(* PLC project Unnamed, Unknown Unnamed 1 *)
(* stored: creationDateTime 2026-04-21T22:15:54, modificationDateTime 2026-04-21T22:15:54 *)

PROGRAM main
  VAR
    input AT %QW0 : INT;
    output AT %QW1 : INT;
  END_VAR

            output := input * 2;
          
END_PROGRAM

CONFIGURATION Config0
  RESOURCE Res0 ON PLC
    TASK task0(INTERVAL := T#20ms, PRIORITY := 1);
    PROGRAM instance0 WITH task0 : main;
  END_RESOURCE
END_CONFIGURATION
